TYPE ST_AXIS_Config :
STRUCT

	sDeviceName				: STRING(30) := 'Axis';
	bCalibrationSensorExist	: BOOL;
	nTorqueLimitation			: UINT	:=	32767;
	stRamps					: ST_AxisCtrlRamps;

END_STRUCT
END_TYPE

(* stored: Version 1.1.0.1, ProductVersion 3.1.4024.15
   DUT ST_AXIS_Config: Id {468d5608-ebaa-45ab-a683-5c6b43b39893} *)
